// TIA Portal V19 export
TYPE "typePosAxisParameter"
// stored: Access Published
   STRUCT
      vel : LReal := 20.0;   // 产品模式设定值，画面做限制根据上限值如果超了不允许输入
      distance : LReal := 10.0;   // 产品模式下拉带走的定长距离
      acc : LReal := 0.5;
      dec : LReal := 0.5;
   END_STRUCT;
END_TYPE
